SYSTEM NonSequentialTest
  (* Version 1.0, 2007-10-25, Goran Cengic, Chalmers *)
  DEVICE Test Device : DeviceType_not_used
    RESOURCE Test Resource : ResourceType_not_used
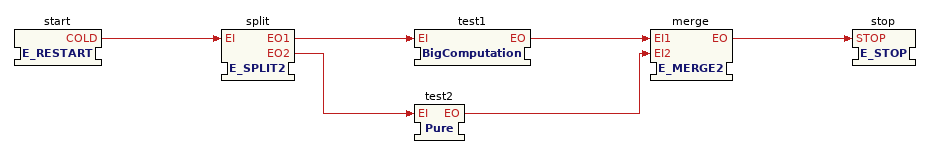
      FBS
        start : E_RESTART;
        split : E_SPLIT2;
        test1 : BigComputation;
        test2 : Pure;
        merge : E_MERGE2;
        stop : E_STOP;
      END_FBS
      EVENT_CONNECTIONS
        start.COLD TO split.EI;
        split.EO1 TO test1.EI;
        split.EO2 TO test2.EI;
        test1.EO TO merge.EI1;
        test2.EO TO merge.EI2;
        merge.EO TO stop.STOP;
      END_CONNECTIONS
    END_RESOURCE
  END_DEVICE
END_SYSTEM
